// Block: RollformingMng_PERS

DATA_BLOCK RollformingMng_PERS
VERSION : 0.1
   NON_RETAIN
   VAR
      PersistentValues : udt_RollformingMng_Pers;
   END_VAR

BEGIN
   // No initialization required
END_DATA_BLOCK
